(* IEC 61131-3 sources: pandora/pandora/aws-platform-main/aws-platform-main/test/Mocks/Io, 4 files *)

(* ---- Digital.st ---- *)
USING Esab.Mock;

NAMESPACE Esab.Io.Mock

    CLASS DigitalInputMock EXTENDS Input IMPLEMENTS IDigitalInput
        VAR PUBLIC
            ReadMock : BoolMethodMock;
            GetValueMock : BoolMethodMock;
            RisingEdgeMock : BoolMethodMock;
            FallingEdgeMock : BoolMethodMock;
            HasChangedMock : BoolMethodMock;
        END_VAR

        METHOD PUBLIC MockReset
            ReadMock.Reset();
            GetValueMock.Reset();
            RisingEdgeMock.Reset();
            FallingEdgeMock.Reset();
            HasChangedMock.Reset();
        END_METHOD

        METHOD PUBLIC Read
            VAR_INPUT
                value : BOOL;
            END_VAR

            ReadMock.IncrementCallCount();
            ReadMock.Value := value;
        END_METHOD

        METHOD PUBLIC GetValue : BOOL
            GetValueMock.IncrementCallCount();
            GetValue := GetValueMock.Value;
        END_METHOD

        METHOD PUBLIC RisingEdge : BOOL
            RisingEdgeMock.IncrementCallCount();
            RisingEdge := RisingEdgeMock.Value;
        END_METHOD

        METHOD PUBLIC FallingEdge : BOOL
            FallingEdgeMock.IncrementCallCount();
            FallingEdge := FallingEdgeMock.Value;
        END_METHOD

        METHOD PUBLIC OVERRIDE HasChanged : BOOL
            HasChangedMock.IncrementCallCount();
            HasChanged := HasChangedMock.Value;
        END_METHOD
    END_CLASS

    CLASS DigitalOutputMock IMPLEMENTS IDigitalOutput
        VAR PUBLIC
            WriteMock : BoolMethodMock;
            SetValueMock : BoolMethodMock;
            SetMock : MethodMock;
            ResetMock : MethodMock;
            ToggleMock : MethodMock;
        END_VAR

        METHOD PUBLIC MockReset
            WriteMock.Reset();
            SetValueMock.Reset();
            SetMock.Reset();
            ResetMock.Reset();
            ToggleMock.Reset();
        END_METHOD

        METHOD PUBLIC Write
            VAR_OUTPUT
                value : BOOL;
            END_VAR

            WriteMock.IncrementCallCount();
            value := WriteMock.Value;
        END_METHOD

        METHOD PUBLIC SetValue
            VAR_INPUT
                value: BOOL;
            END_VAR

            SetValueMock.IncrementCallCount();
            SetValueMock.Value := value;
        END_METHOD

        METHOD PUBLIC Set
            SetMock.IncrementCallCount();
        END_METHOD

        METHOD PUBLIC Reset
            ResetMock.IncrementCallCount();
        END_METHOD

        METHOD PUBLIC Toggle
            ToggleMock.IncrementCallCount();
        END_METHOD
    END_CLASS

END_NAMESPACE

(* ---- DInt.st ---- *)
USING Esab.Mock;

NAMESPACE Esab.Io.Mock

    CLASS DIntInputMock EXTENDS Input IMPLEMENTS IDIntInput
        VAR PUBLIC
            ReadMock : DIntMethodMock;
            GetValueMock : DIntMethodMock;
            HasChangedMock : BoolMethodMock;
        END_VAR

        METHOD PUBLIC MockReset
            ReadMock.Reset();
            GetValueMock.Reset();
        END_METHOD

        METHOD PUBLIC Read
            VAR_INPUT
                value : DINT;
            END_VAR

            ReadMock.IncrementCallCount();
            ReadMock.Value := value;
        END_METHOD

        METHOD PUBLIC GetValue : DINT
            GetValueMock.IncrementCallCount();
            GetValue := GetValueMock.Value;
        END_METHOD

        METHOD PUBLIC OVERRIDE HasChanged : BOOL
            HasChangedMock.IncrementCallCount();
            HasChanged := HasChangedMock.Value;
        END_METHOD
    END_CLASS

    CLASS DintOutputMock IMPLEMENTS IDintOutput
        VAR PUBLIC
            WriteMock : DIntMethodMock;
            SetValueMock : DIntMethodMock;
            SetMock : MethodMock;
            ResetMock : MethodMock;
            ToggleMock : MethodMock;
        END_VAR

        METHOD PUBLIC MockReset
            WriteMock.Reset();
            SetValueMock.Reset();
            SetMock.Reset();
            ResetMock.Reset();
            ToggleMock.Reset();
        END_METHOD

        METHOD PUBLIC Write
            VAR_OUTPUT
                value : DINT;
            END_VAR

            WriteMock.IncrementCallCount();
            value := WriteMock.Value;
        END_METHOD

        METHOD PUBLIC SetValue
            VAR_INPUT
                value: DINT;
            END_VAR

            SetValueMock.IncrementCallCount();
            SetValueMock.Value := value;
        END_METHOD

        METHOD PUBLIC Set
            SetMock.IncrementCallCount();
        END_METHOD

        METHOD PUBLIC Reset
            ResetMock.IncrementCallCount();
        END_METHOD

        METHOD PUBLIC Toggle
            ToggleMock.IncrementCallCount();
        END_METHOD
    END_CLASS

END_NAMESPACE

(* ---- UInt.st ---- *)
USING Esab.Mock;

NAMESPACE Esab.Io.Mock

    CLASS UIntInputMock EXTENDS Input IMPLEMENTS IUIntInput
        VAR PUBLIC
            ReadUIntMock : UIntMethodMock;
            ReadByteMock : ByteMethodMock;
            GetValueMock : UIntMethodMock;
            HasChangedMock : BoolMethodMock;
        END_VAR

        METHOD PUBLIC MockReset
            ReadUIntMock.Reset();
            ReadByteMock.Reset();
            GetValueMock.Reset();
            HasChangedMock.Reset();
        END_METHOD

        METHOD PUBLIC Read
            VAR_INPUT
                value : UINT;
            END_VAR

            ReadUIntMock.IncrementCallCount();
            ReadUIntMock.Value := value;
        END_METHOD

        METHOD PUBLIC Read
            VAR_INPUT
                value : BYTE;
            END_VAR

            ReadByteMock.IncrementCallCount();
            ReadByteMock.Value := value;
        END_METHOD

        METHOD PUBLIC GetValue : UINT
            GetValueMock.IncrementCallCount();
            GetValue := GetValueMock.Value;
        END_METHOD

        METHOD PUBLIC OVERRIDE HasChanged : BOOL
            HasChangedMock.IncrementCallCount();
            HasChanged := HasChangedMock.Value;
        END_METHOD
    END_CLASS

    CLASS UIntOutputMock IMPLEMENTS IUIntOutput
        VAR PUBLIC
            WriteUIntMock : UIntMethodMock;
            WriteByteMock : ByteMethodMock;
            SetValueUIntMock : UIntMethodMock;
            SetValueByteMock : ByteMethodMock;
            SetMock : MethodMock;
            ResetMock : MethodMock;
            ToggleMock : MethodMock;
        END_VAR

        METHOD PUBLIC MockReset
            WriteUIntMock.Reset();
            WriteByteMock.Reset();
            SetValueUIntMock.Reset();
            SetValueByteMock.Reset();
            SetMock.Reset();
            ResetMock.Reset();
            ToggleMock.Reset();
        END_METHOD

        METHOD PUBLIC Write
            VAR_OUTPUT
                value : UINT;
            END_VAR

            WriteUIntMock.IncrementCallCount();
            value := WriteUIntMock.Value;
        END_METHOD

        METHOD PUBLIC Write
            VAR_OUTPUT
                value : BYTE;
            END_VAR

            WriteByteMock.IncrementCallCount();
            value := WriteByteMock.Value;
        END_METHOD

        METHOD PUBLIC SetValue
            VAR_INPUT
                value: UINT;
            END_VAR

            SetValueUIntMock.IncrementCallCount();
            SetValueUIntMock.Value := value;
        END_METHOD

        METHOD PUBLIC SetValue
            VAR_INPUT
                value: BYTE;
            END_VAR

            SetValueByteMock.IncrementCallCount();
            SetValueByteMock.Value := value;
        END_METHOD

        METHOD PUBLIC Set
            SetMock.IncrementCallCount();
        END_METHOD

        METHOD PUBLIC Reset
            ResetMock.IncrementCallCount();
        END_METHOD

        METHOD PUBLIC Toggle
            ToggleMock.IncrementCallCount();
        END_METHOD
    END_CLASS

END_NAMESPACE

(* ---- Io.st ---- *)
NAMESPACE Esab.Io.Mock
END_NAMESPACE
